FUNCTION_BLOCK EQ_Scale (* Scale; the hardware has none yet (the ESP32 publishes a random weight), so it is simulated; equipment IO: owns its IO points; commands Idle=0, Tare=1, Measure=2 *)
  (* Standard: 61499-2 *)
  (* Version 0.1, 2026-09-28, Project contributors, AAU Smart Production Lab *)
  PACKAGE filling;
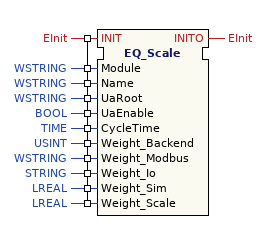
  EVENT_INPUT
    INIT : EInit WITH Module, Name, UaRoot, UaEnable, CycleTime, Weight_Backend, Weight_Modbus, Weight_Io, Weight_Sim, Weight_Scale;
  END_EVENT
  EVENT_OUTPUT
    INITO : EInit;
  END_EVENT
  VAR_INPUT
    Module : WSTRING;
    Name : WSTRING := "Scale";
    UaRoot : WSTRING;
    UaEnable : BOOL;
    CycleTime : TIME := T#50ms;
    Weight_Backend : USINT := 2;
    Weight_Modbus : WSTRING;
    Weight_Io : STRING;
    Weight_Sim : LREAL := 2.0;
    Weight_Scale : LREAL := 0.001;
  END_VAR
  FBS
    Logic : filling::EL_Scale;
    Mode : modlib::MOD_StateView;
    SubCmd : iec61499::net::SUBSCRIBE_4(QI := TRUE);
    PubState : iec61499::net::PUBLISH_2(QI := TRUE);
    PubUa : iec61499::net::PUBLISH_1;
    In_Weight : modlib::IO_AI;
    Cycle : iec61499::events::E_CYCLE;
    PhaseT : iec61499::events::E_DELAY;
  END_FBS
  EVENT_CONNECTIONS
    INIT TO Logic.INIT;
    Logic.INITO TO Mode.INIT;
    Mode.INITO TO SubCmd.INIT;
    SubCmd.INITO TO PubState.INIT;
    PubState.INITO TO PubUa.INIT;
    PubUa.INITO TO In_Weight.INIT;
    In_Weight.INITO TO Cycle.START;
    In_Weight.INITO TO INITO;
    SubCmd.IND TO Logic.CMD;
    Mode.CHG TO Logic.MOD_CHG;
    Cycle.EO TO Logic.REFRESH;
    Cycle.EO TO In_Weight.REQ;
    In_Weight.CNF TO Logic.SAMPLE;
    Logic.STATE TO PubState.REQ;
    Logic.STATE TO PubUa.REQ;
    Logic.DRIVE TO Logic.DRIVEN;
    Logic.PHASE_START TO PhaseT.START;
    Logic.PHASE_STOP TO PhaseT.STOP;
    PhaseT.EO TO Logic.PHASE_T;
  END_CONNECTIONS
  DATA_CONNECTIONS
    Module TO Logic.Module;
    Name TO Logic.Name;
    UaRoot TO Logic.UaRoot;
    Module TO Mode.Module;
    Logic.IdCmd TO SubCmd.ID;
    Logic.IdState TO PubState.ID;
    Logic.IdPub TO PubUa.ID;
    UaEnable TO PubUa.QI;
    CycleTime TO Cycle.DT;
    SubCmd.RD_1 TO Logic.C_Holder;
    SubCmd.RD_2 TO Logic.C_Command;
    SubCmd.RD_3 TO Logic.C_Arg;
    SubCmd.RD_4 TO Logic.C_Release;
    Mode.State TO Logic.ModState;
    Weight_Backend TO In_Weight.Backend;
    Weight_Modbus TO In_Weight.ModbusId;
    Weight_Io TO In_Weight.IoName;
    Weight_Sim TO In_Weight.SimValue;
    Weight_Scale TO In_Weight.Scale;
    In_Weight.IN TO Logic.I_Weight;
    Logic.Weight TO PubState.SD_1;
    Logic.Weight TO PubUa.SD_1;
    Logic.Holder TO PubState.SD_2;
    Logic.PhaseDT TO PhaseT.DT;
  END_CONNECTIONS
END_FUNCTION_BLOCK
